// TIA Portal V20 export
TYPE "LER_typeSoftCamInterface2"
// stored: Access Published
   STRUCT
      pos0 { S7_SetPoint := 'True'} : "LER_typeSoftcamControlNodes";
      pos1 { S7_SetPoint := 'True'} : "LER_typeSoftcamControlNodes";
      pos2 { S7_SetPoint := 'True'} : "LER_typeSoftcamControlNodes";
      pos3 { S7_SetPoint := 'True'} : "LER_typeSoftcamControlNodes";
      pos4 { S7_SetPoint := 'True'} : "LER_typeSoftcamControlNodes";
      pos5 { S7_SetPoint := 'True'} : "LER_typeSoftcamControlNodes";
      pos6 { S7_SetPoint := 'True'} : "LER_typeSoftcamControlNodes";
      pos7 { S7_SetPoint := 'True'} : "LER_typeSoftcamControlNodes";
      pos8 { S7_SetPoint := 'True'} : "LER_typeSoftcamControlNodes";
      pos9 { S7_SetPoint := 'True'} : "LER_typeSoftcamControlNodes";
      pos10 { S7_SetPoint := 'True'} : "LER_typeSoftcamControlNodes";
      pos11 { S7_SetPoint := 'True'} : "LER_typeSoftcamControlNodes";
      pos12 { S7_SetPoint := 'True'} : "LER_typeSoftcamControlNodes";
      pos13 { S7_SetPoint := 'True'} : "LER_typeSoftcamControlNodes";
      pos14 { S7_SetPoint := 'True'} : "LER_typeSoftcamControlNodes";
      pos15 { S7_SetPoint := 'True'} : "LER_typeSoftcamControlNodes";
   END_STRUCT;
END_TYPE
